// This function has been automatically generated from the project information.
{attribute 'signature_flag' := '1073741824'}
{attribute 'TcGenerated'}
{attribute 'no-analysis'}
FUNCTION F_GetCompany : WSTRING
VAR_INPUT
	
END_VAR

F_GetCompany := "BA Belgium";

END_FUNCTION

(* stored: Version 1.1.0.1
   POU F_GetCompany: Id {0614a653-f08f-4247-9c39-28094ceea9a9}, SpecialFunc None *)
